FUNCTION_BLOCK FB_HandleUiEstop
VAR_INPUT
	button : BOOL;
	reset : BOOL;
END_VAR
VAR_OUTPUT
	stop : BOOL;
END_VAR
VAR
	RTRIG_ButtonPressed : R_TRIG;
	RTRIG_resetPressed : R_TRIG;
END_VAR


RTRIG_ButtonPressed(CLK := button);
IF RTRIG_ButtonPressed.Q THEN
	stop := TRUE;
END_IF

RTRIG_resetPressed(CLK := reset);
IF RTRIG_resetPressed.q THEN
	stop := FALSE;
END_IF

END_FUNCTION_BLOCK

(* stored: Version 1.1.0.1, ProductVersion 3.1.4024.9
   POU FB_HandleUiEstop: Id {494017d8-bd6a-437d-bc9e-5e9024c1895e}, SpecialFunc None *)
